SUBAPPLICATION Checkbox_IDA_TO_AX (* VT-Checkbox live als AX (Pegel) weiterreichen (isobus::UT::io::NumericValue::NumericValue_IDA + AD_TO_AX), reiner Ein/Aus-Zustand ohne Skalierung/Persistenz, z.B. fuer Automatik_Toggle.PERMIT. WICHTIG: u16ObjId ist die ObjectID der CNumberVariable, die die Checkbox als Wertspeicher referenziert (z.B. NumberVariable_Bunker_Fuellstand_Hoehe_Automatik) - NICHT die ObjectID der Checkbox (CInputBoolean) selbst, die VT meldet Value-Aenderungen unter der NumberVariable-ID (Franz, live verifiziert). *)
  (* Standard: 61499-2; Description: Copyright (c) 2026 Meisterschulen am Ostbahnhof This program and the accompanying materials are made available under the terms of the Eclipse Public License 2.0 which is available at https://www.eclipse.org/legal/epl-2.0/ SPDX-License-Identifier: EPL-2.0 *)
  (* Version 1.0, 2026-09-27, Franz Höpfinger, Meisterschulen am Ostbahnhof, initial implementation - Franz: 'NumberVariable_Bunker_Fuellstand_Hoehe_Automatik soll das GESAMTE AN/Aus der Befuellautomatik gaten, wirkt wie ein AX_PERMIT' - liest die neue VT-Checkbox (InputBoolean) roh per ObjectID via NumericValue_IDA (AD) + AD_TO_AX (DWORD<>0), fuer Automatik_Toggle.PERMIT. *)
  PACKAGE MyLib::sys;
  IMPORT isobus::UT::Q::const::IDs::ID_NULL;
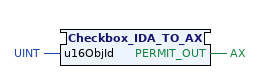
  VAR_INPUT
    u16ObjId : UINT := ID_NULL; (* Object ID der VT-Checkbox (InputBoolean) *)
  END_VAR
  PLUGS
    PERMIT_OUT : adapter::types::unidirectional::AX; (* Roher Checkbox-Zustand (0/1) als Pegel *)
  END_PLUGS
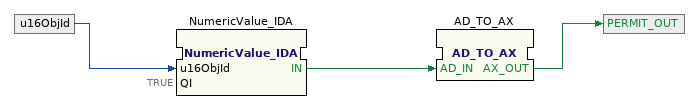
  FBS
    NumericValue_IDA : isobus::UT::io::NumericValue::NumericValue_IDA(QI := TRUE);
    AD_TO_AX : adapter::conversion::unidirectional::AD_TO_AX;
  END_FBS
  DATA_CONNECTIONS
    u16ObjId TO NumericValue_IDA.u16ObjId;
  END_CONNECTIONS
  ADAPTER_CONNECTIONS
    NumericValue_IDA.IN TO AD_TO_AX.AD_IN;
    AD_TO_AX.AX_OUT TO PERMIT_OUT;
  END_CONNECTIONS
END_SUBAPPLICATION
